FUNCTION_BLOCK FB_InitChecks
VAR_INPUT
	bPower24V_OK : BOOL;
    bPower48V_OK : BOOL;
    bDoorsClosed : BOOL;
    bDoorsLocked : BOOL;
    bAirEnabled  : BOOL;
END_VAR
VAR_OUTPUT
	bInitOK : BOOL; 	//Indicates whether you can advance from one state to another
    bError  : BOOL;
END_VAR
VAR
	fbEventHandler : FB_EventHandler;
    bExecuteEvent  : BOOL := FALSE;
    bEventDone     : BOOL := FALSE;
END_VAR

// 1. Check the power supply
IF NOT (bPower24V_OK AND bPower48V_OK) THEN
    bError := TRUE;
    bExecuteEvent := TRUE;
    fbEventHandler(
        bExecute  := bExecuteEvent,
        eEventName := E_Events.ERROR,
        sSystem    := 'Power Supply Check',
        sMessage   := 'Power Supply 24/48Vdc with Error!',
        bDone      => bEventDone
    );
    ResetEventTrigger();
    
    //Reset air supply and door lock commands
    GVL_Safety.bAirSupplyEnable := FALSE;
    GVL_Safety.bDoorLockCommand := FALSE;

// 2. Check if doors are closed
ELSIF NOT bDoorsClosed THEN
    bExecuteEvent := TRUE;
    fbEventHandler(
        bExecute  := bExecuteEvent,
        eEventName := E_Events.WARNING,
        sSystem    := 'Safety',
        sMessage   := 'Doors not closed!',
        bDone      => bEventDone
    );
    ResetEventTrigger();

    //Reset air supply and door lock commands
    GVL_Safety.bAirSupplyEnable := FALSE;
    GVL_Safety.bDoorLockCommand := FALSE;

// 3. Lock doors if they are not locked
ELSIF NOT bDoorsLocked THEN
    GVL_Safety.bDoorLockCommand := TRUE; //Lock the doors

    //Reset air supply command
    GVL_Safety.bAirSupplyEnable := FALSE;

// 4. If doors are locked but air is not enabled, activate air supply
ELSIF NOT bAirEnabled THEN
    bExecuteEvent := TRUE;
    fbEventHandler(
        bExecute  := bExecuteEvent,
        eEventName := E_Events.INFO,
        sSystem    := 'Safety',
        sMessage   := 'All Doors Locked!',
        bDone      => bEventDone
    );
    ResetEventTrigger();
	
    GVL_Safety.SafetyOutputs.bAirPressureOK := TRUE; //#TODO meassuring the airsupply
    GVL_Safety.bAirSupplyEnable := TRUE;

// 5. If everything is OK, move to the next state
ELSE
    bExecuteEvent := TRUE;
    fbEventHandler(
        bExecute  := bExecuteEvent,
        eEventName := E_Events.INFO,
        sSystem    := 'Safety',
        sMessage   := 'Air Supply Enabled!',
        bDone      => bEventDone
    );
    ResetEventTrigger();
    
    bInitOK := TRUE;
END_IF;

ACTION ResetEventTrigger:
IF bEventDone THEN
        bExecuteEvent := FALSE;
        bEventDone := FALSE;
END_IF;
END_ACTION

END_FUNCTION_BLOCK

(* stored: Version 1.1.0.1, ProductVersion 3.1.4024.12
   POU FB_InitChecks: Id {ca2f8e73-30a6-41b7-a1d5-e28e096b5f8e}, SpecialFunc None
   Action ResetEventTrigger: Id {ddb8bc5a-944b-470b-9118-654fa8c992ef} *)
